Staubli VAL3: start.pgx

program start()
  local num l_nCounter
  local num l_nLatched
  local bool l_bLatched
begin
  cls()
  userPage()
  call create(0,"encoder")
  do
    call isLatched(l_bLatched)
    if l_bLatched==true
      call getValue(false,l_nCounter)
      call getValue(true,l_nLatched)
      gotoxy(0,10)
      putln(l_nCounter)
      gotoxy(20,10)
      putln(l_nLatched)
    endIf
    delay(0)
  until false
end
